// TIA Portal V17 export
// export: Created 2025-06-26T06:33:59.5579082Z, ExportSetting WithDefaults, DisplayName Totally Integrated Automation Portal, DisplayVersion V17 Update 8, DisplayName TIA Portal Openness, DisplayVersion V17 Update 8, DisplayName TIA Portal Version Control Interface, DisplayVersion V17, DisplayName STEP 7 Professional, DisplayVersion V17 Update 8, DisplayName STEP 7 Safety, DisplayVersion V17 Update 6, DisplayName WinCC Advanced, DisplayVersion V17 Update 8
VAR_GLOBAL   // PLC tag table "Local_IO"
   DQa_0 AT %Q0.0 : Bool;
   DQa_1 AT %Q0.1 : Bool;
   DQa_2 AT %Q0.2 : Bool;
   DQa_3 AT %Q0.3 : Bool;
   DQa_4 AT %Q0.4 : Bool;
   DQa_5 AT %Q0.5 : Bool;
   DQa_6 AT %Q0.6 : Bool;
   DQa_7 AT %Q0.7 : Bool;
   DQb_0 AT %Q1.0 : Bool;
   DQb_1 AT %Q1.1 : Bool;
   DIa_0 AT %I0.0 : Bool;
   DIa_1 AT %I0.1 : Bool;
   DIa_2 AT %I0.2 : Bool;
   DIa_3 AT %I0.3 : Bool;
   DIa_4 AT %I0.4 : Bool;
   DIa_5 AT %I0.5 : Bool;
   DIa_6 AT %I0.6 : Bool;
   DIa_7 AT %I0.7 : Bool;
   DIb_0 AT %I1.0 : Bool;
   DIb_1 AT %I1.1 : Bool;
   DIb_2 AT %I1.2 : Bool;
   DIb_3 AT %I1.3 : Bool;
   DIb_4 AT %I1.4 : Bool;
   DIb_5 AT %I1.5 : Bool;
END_VAR
